(*

.. <legal notes>

legal notes
=================
| SPDX-FileCopyrightText: © 2025 Oleksandr Tiutyk <trofimich@gmail.com>
| SPDX-License-Identifier: LGPL-3.0-only
| For details check: LGPL-3.0-only_

.. _LGPL-3.0-only: https://www.gnu.org/licenses/lgpl-3.0.en.html

.. </legal notes>

*)

{attribute 'no_explicit_call' := 'do not call this function block directly'} 
FUNCTION_BLOCK ABSTRACT Task EXTENDS Object IMPLEMENTS ITask
VAR
	_Name : WSTRING;
	
	_StateChanged : BOOL;

	_Busy : BOOL;
	
	_Done : BOOL;

	_Cancelled : BOOL;
	
	_Aborted : BOOL;
	
	_Error : BOOL;	
	_ErrorMessage : ERROR_MESSAGE;	
END_VAR

{attribute 'monitoring' := 'call'}
{attribute 'OPC.UA.DA.Property' := '1'}
{attribute 'OPC.UA.DA.Access' := '1'}
PROPERTY FINAL Aborted : BOOL
GET
Aborted := _Aborted;
END_GET
END_PROPERTY

{attribute 'monitoring' := 'call'}
{attribute 'OPC.UA.DA.Property' := '1'}
{attribute 'OPC.UA.DA.Access' := '1'}
PROPERTY FINAL Busy : BOOL
GET
Busy := _Busy;
END_GET
END_PROPERTY

METHOD FINAL Cancel
VAR
	exceptionCode : __SYSTEM.ExceptionCode;
	
	exception : IException;
END_VAR
IF Busy THEN
	RETURN;
END_IF

__TRY
	OnCancel();
	
	setCancelledState();
__CATCH(exceptionCode)
	handleFault(exceptionCode);
__ENDTRY
END_METHOD

{attribute 'monitoring' := 'call'}
{attribute 'OPC.UA.DA.Property' := '1'}
{attribute 'OPC.UA.DA.Access' := '1'}
PROPERTY FINAL Cancelled : BOOL
GET
Cancelled := _Cancelled;
END_GET
END_PROPERTY

{attribute 'monitoring' := 'call'}
{attribute 'OPC.UA.DA.Property' := '1'}
{attribute 'OPC.UA.DA.Access' := '1'}
PROPERTY FINAL Done : BOOL
GET
Done := _Done OR_ELSE _Aborted OR_ELSE _Error;
END_GET
END_PROPERTY

{attribute 'monitoring' := 'call'}
{attribute 'OPC.UA.DA.Property' := '1'}
{attribute 'OPC.UA.DA.Access' := '1'}
PROPERTY FINAL Error : BOOL
GET
Error := _Error;
END_GET
END_PROPERTY

{attribute 'monitoring' := 'call'}
{attribute 'OPC.UA.DA.Property' := '1'}
{attribute 'OPC.UA.DA.Access' := '1'}
PROPERTY FINAL ErrorMessage : REFERENCE TO ERROR_MESSAGE
GET
ErrorMessage REF= _ErrorMessage;
END_GET
END_PROPERTY

METHOD FINAL Execute 
VAR
	runningState : TASK_RUNNING_STATE;
	
	exceptionCode : __SYSTEM.ExceptionCode;
	
	exception : IException;	
	
	errorMessage : ERROR_MESSAGE;
END_VAR
_StateChanged := FALSE;

__TRY
	IF Busy THEN
		OnRunning(FALSE, state => runningState);
		
		CASE runningState OF
			TASK_RUNNING_STATE.DONE:
				setDoneState();
			
			TASK_RUNNING_STATE.ABORTED:
				setAbortedState();
		END_CASE
	END_IF
__CATCH(exceptionCode)
	handleFault(exceptionCode);
__ENDTRY
END_METHOD

METHOD PRIVATE handleFault
VAR_INPUT
	exceptionCode : __SYSTEM.ExceptionCode;
END_VAR
VAR
	exception : IException;
END_VAR
exception := ExceptionManager.GetLastException(exceptionCode);

__TRY
	OnFault();
__CATCH
__ENDTRY
	
IF NOT _Error THEN
	LogManager.TryLogMessage(WideStringHelper.ConcatStrings255("Task '", Name, "' failed at ", TO_WSTRING(SystemDateTimeManager.SystemLocalDateTime)), LOG_CATEGORY.SUCCESS, TO_WSTRING(ClassName), "Task", "TaskError");
	
	_StateChanged := TRUE;
END_IF

_Busy := FALSE;

_Done := FALSE;

_Cancelled := FALSE;

_Aborted := FALSE;

_Error := TRUE;		
_ErrorMessage := exception.GetMessage();

ExceptionManager.Throw(exception);
END_METHOD

{attribute 'monitoring' := 'call'}
{attribute 'OPC.UA.DA.Property' := '1'}
{attribute 'OPC.UA.DA.Access' := '1'}
PROPERTY FINAL Name : WSTRING
GET
Name := SEL(_Name = "", _Name, SUPER^.Name);
END_GET
SET
_Name := Name;
END_SET
END_PROPERTY

METHOD PROTECTED ABSTRACT OnCancel
END_METHOD

METHOD PROTECTED OnFault
END_METHOD

METHOD PROTECTED ABSTRACT OnRunning 
VAR_INPUT
	startRequest : BOOL;
END_VAR
VAR_OUTPUT
	state : TASK_RUNNING_STATE;
END_VAR
END_METHOD

METHOD PRIVATE FINAL setAbortedState
IF NOT _Aborted THEN
	LogManager.TryLogMessage(WideStringHelper.ConcatStrings255("Task '", Name, "' aborted at ", TO_WSTRING(SystemDateTimeManager.SystemLocalDateTime)), LOG_CATEGORY.SUCCESS, TO_WSTRING(ClassName), "Task", "TaskAborted");

	_StateChanged := TRUE;
END_IF

_Busy := FALSE;

_Done := FALSE;

_Cancelled := FALSE;

_Aborted := TRUE;

_Error := FALSE;	
_ErrorMessage := "";
END_METHOD

METHOD PRIVATE FINAL setBusyState
IF NOT _Busy THEN
	LogManager.TryLogMessage(WideStringHelper.ConcatStrings255("Task '", Name, "' started at ", TO_WSTRING(SystemDateTimeManager.SystemLocalDateTime)), LOG_CATEGORY.SUCCESS, TO_WSTRING(ClassName), "Task", "TaskBusy");
	
	_StateChanged := TRUE;
END_IF

_Busy := TRUE;

_Done := FALSE;

_Cancelled := FALSE;

_Aborted := FALSE;

_Error := FALSE;	
_ErrorMessage := "";
END_METHOD

METHOD PRIVATE FINAL setCancelledState
IF NOT _Aborted THEN
	LogManager.TryLogMessage(WideStringHelper.ConcatStrings255("Task '", Name, "' cancelled at ", TO_WSTRING(SystemDateTimeManager.SystemLocalDateTime)), LOG_CATEGORY.SUCCESS, TO_WSTRING(ClassName), "Task", "TaskCancelled");

	_StateChanged := TRUE;
END_IF

_Busy := FALSE;

_Done := FALSE;

_Cancelled := TRUE;

_Aborted := FALSE;

_Error := FALSE;	
_ErrorMessage := "";
END_METHOD

METHOD PRIVATE FINAL setDoneState
IF NOT _Done THEN
	LogManager.TryLogMessage(WideStringHelper.ConcatStrings255("Task '", Name, "' done at ", TO_WSTRING(SystemDateTimeManager.SystemLocalDateTime)), LOG_CATEGORY.SUCCESS, TO_WSTRING(ClassName), "Task", "TaskDone");
	
	_StateChanged := TRUE;
END_IF

_Busy := FALSE;

_Done := TRUE;

_Cancelled := FALSE;

_Aborted := FALSE;

_Error := FALSE;	
_ErrorMessage := "";
END_METHOD

METHOD FINAL Start : BOOL
VAR
	runningState : TASK_RUNNING_STATE;

	exceptionCode : __SYSTEM.ExceptionCode;
	
	exception : IException;
END_VAR
IF Busy THEN
	RETURN;
END_IF

__TRY
	setBusyState();
	
	OnRunning(TRUE, state => runningState);

	CASE runningState OF
		TASK_RUNNING_STATE.DONE:
			setDoneState();
		
		TASK_RUNNING_STATE.ABORTED:
			setAbortedState();	
	END_CASE
	
	Start := TRUE;
__CATCH(exceptionCode)
	handleFault(exceptionCode);
__ENDTRY
END_METHOD

{attribute 'monitoring' := 'call'}
{attribute 'OPC.UA.DA.Property' := '1'}
{attribute 'OPC.UA.DA.Access' := '1'}
PROPERTY FINAL StateChanged : BOOL
GET
StateChanged := _StateChanged;
END_GET
END_PROPERTY

END_FUNCTION_BLOCK

(* stored: Version 1.1.0.1
   POU Task: Id {3fcb82bf-fcc2-4c60-ab58-32776172ce5b}, SpecialFunc None
   Folder Members to override: Id {76112447-5878-4246-92fb-0910ffa3ef2d}
   Folder Service members: Id {6b1a5589-8d7c-4542-877b-5fcd2d9b2fbd}
   Property Aborted: Id {205fba08-26d2-4312-a96e-e17dee6c923f}
   Get Get: Id {9f8851fa-4d24-41c2-b7cf-fd9ecc9bdb84}
   Property Busy: Id {e3f55a84-6dc8-42a8-870b-cbc03d5ce896}
   Get Get: Id {9b0f9833-3b49-48b8-9041-0090b996669f}
   Method Cancel: Id {85ebde85-30ac-4488-ad53-ac1ecdb74776}
   Property Cancelled: Id {72ad9134-a921-4460-953e-dd085c603cb7}
   Get Get: Id {6008e232-f65d-448f-8b7c-75b411e44c3a}
   Property Done: Id {10c3e2b7-99f3-4fa9-bdac-62a94dfa4509}
   Get Get: Id {bbb5f7ba-4447-4958-8ec9-7e3859b0437b}
   Property Error: Id {3d54590f-9d24-46b4-9724-32260ce4207a}
   Get Get: Id {998b8321-1744-4a0a-b9cf-78a20c7dc6e5}
   Property ErrorMessage: Id {e92b95ec-4a2f-46a9-85eb-1f48df75a257}
   Get Get: Id {82e42fe0-1017-4cc0-a630-23020b73322e}
   Method Execute: Id {356dfaf1-5836-4634-88c3-9adf266fe2b8}
   Method handleFault: Id {87f22517-b446-496a-a773-92d534ab21f6}
   Property Name: Id {82c59c7f-12d8-4fab-8d33-ec1ebb7c64fc}
   Get Get: Id {61eb0fbe-e691-4c63-b864-dbfd0811101b}
   Set Set: Id {8648b17d-3897-46ca-b930-e499fe043a7b}
   Method OnCancel: Id {e62e6e28-d2f5-4a49-a4f3-1ac1c3a6c40e}
   Method OnFault: Id {c12cd4b4-6b5e-40a4-9547-4538d1fad656}
   Method OnRunning: Id {a15599f5-e9ad-4bc1-b827-e975fc966d86}
   Method setAbortedState: Id {fac00809-31d6-4f90-8e02-b442214ce266}
   Method setBusyState: Id {8ba032d1-b467-4f29-94d8-e5d440995321}
   Method setCancelledState: Id {9eb02e57-605e-46fb-afde-513fb736d90a}
   Method setDoneState: Id {5a91bd28-905f-4ff0-ac15-4afd240589a6}
   Method Start: Id {5e4f958e-3441-449c-a3ee-2bfa2bc2b0b1}
   Property StateChanged: Id {5df375fb-8678-4172-86a8-056cc8dfa2cd}
   Get Get: Id {68fadd26-a99e-461e-8aa1-2b482d0dd654} *)
